PROGRAM Intfc_Upstream_ML
VAR
	Upstream_Upper_LaneA_Comm		: FB_ReadAdsSymByName;
	Upstream_Upper_LaneB_Comm		: FB_ReadAdsSymByName;
	Upstream_Upper_ExitLane_Comm	: FB_ReadAdsSymByName;
	Upstream_Lower_LaneA_Comm		: FB_ReadAdsSymByName;
	Upstream_Lower_LaneB_Comm		: FB_ReadAdsSymByName;
	Upstream_Lower_ExitLane_Comm	: FB_ReadAdsSymByName;
	UpdateRate						: TIME;
	UpdateTimer						: TON;
	UpdateCounter					: CTU;
END_VAR

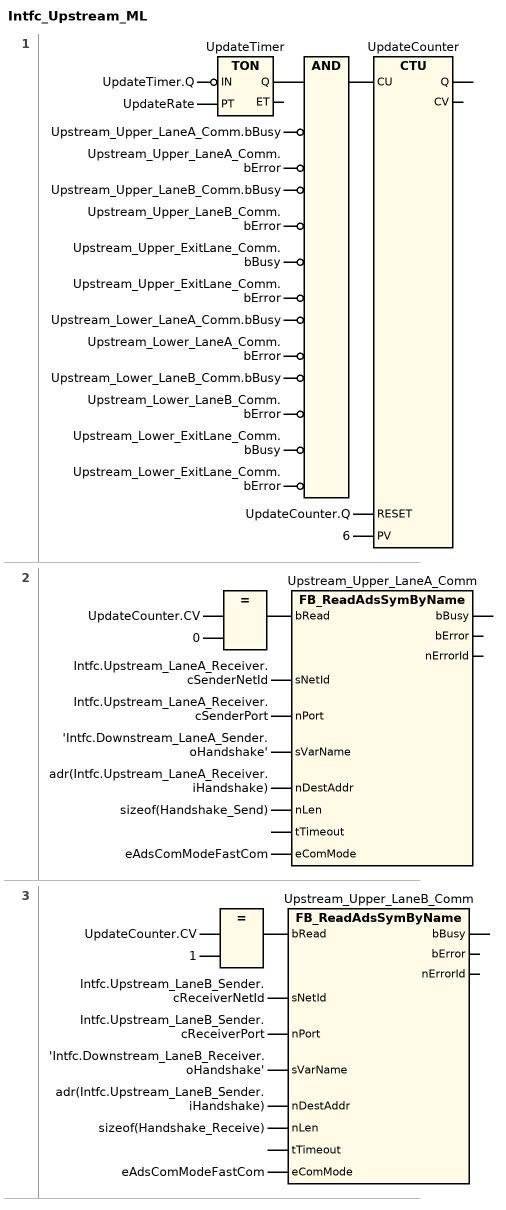
// NETWORK 1
UpdateTimer(IN := NOT UpdateTimer.Q, PT := UpdateRate); // TON
UpdateCounter(
    CU := UpdateTimer.Q AND NOT Upstream_Upper_LaneA_Comm.bBusy AND NOT Upstream_Upper_LaneA_Comm.bError AND NOT Upstream_Upper_LaneB_Comm.bBusy AND NOT Upstream_Upper_LaneB_Comm.bError AND NOT Upstream_Upper_ExitLane_Comm.bBusy AND NOT Upstream_Upper_ExitLane_Comm.bError AND NOT Upstream_Lower_LaneA_Comm.bBusy AND NOT Upstream_Lower_LaneA_Comm.bError AND NOT Upstream_Lower_LaneB_Comm.bBusy AND NOT Upstream_Lower_LaneB_Comm.bError AND NOT Upstream_Lower_ExitLane_Comm.bBusy AND NOT Upstream_Lower_ExitLane_Comm.bError,
    RESET := UpdateCounter.Q,
    PV := 6); // CTU

// NETWORK 2
Upstream_Upper_LaneA_Comm(
    bRead := UpdateCounter.CV = 0,
    sNetId := Intfc.Upstream_LaneA_Receiver.cSenderNetId,
    nPort := Intfc.Upstream_LaneA_Receiver.cSenderPort,
    sVarName := 'Intfc.Downstream_LaneA_Sender.oHandshake',
    nDestAddr := adr(Intfc.Upstream_LaneA_Receiver.iHandshake),
    nLen := sizeof(Handshake_Send),
    eComMode := eAdsComModeFastCom); // FB_ReadAdsSymByName

// NETWORK 3
Upstream_Upper_LaneB_Comm(
    bRead := UpdateCounter.CV = 1,
    sNetId := Intfc.Upstream_LaneB_Sender.cReceiverNetId,
    nPort := Intfc.Upstream_LaneB_Sender.cReceiverPort,
    sVarName := 'Intfc.Downstream_LaneB_Receiver.oHandshake',
    nDestAddr := adr(Intfc.Upstream_LaneB_Sender.iHandshake),
    nLen := sizeof(Handshake_Receive),
    eComMode := eAdsComModeFastCom); // FB_ReadAdsSymByName

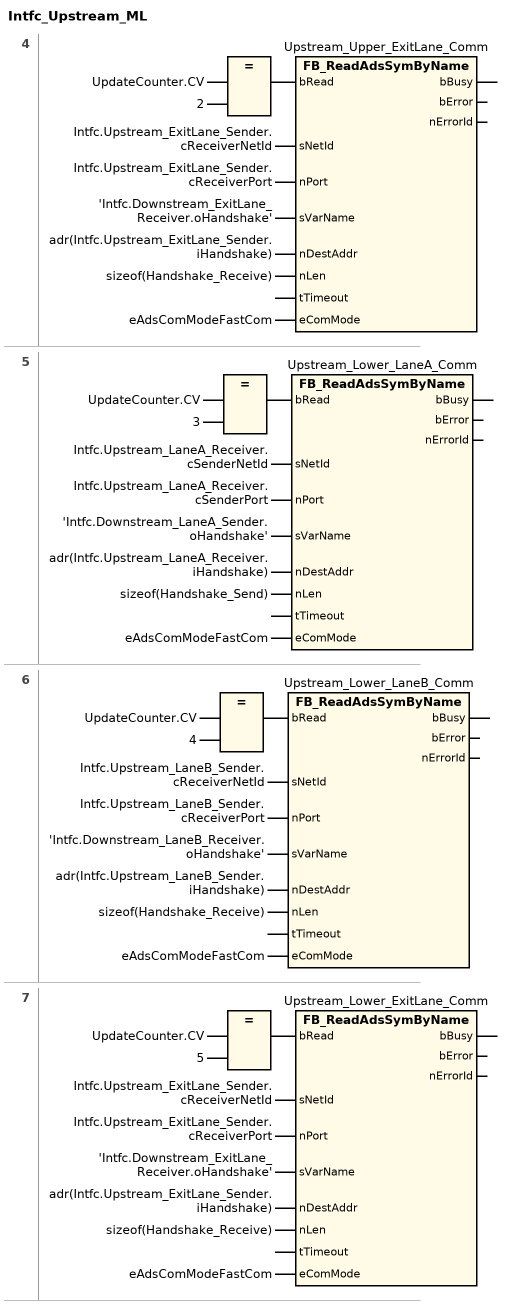
// NETWORK 4
Upstream_Upper_ExitLane_Comm(
    bRead := UpdateCounter.CV = 2,
    sNetId := Intfc.Upstream_ExitLane_Sender.cReceiverNetId,
    nPort := Intfc.Upstream_ExitLane_Sender.cReceiverPort,
    sVarName := 'Intfc.Downstream_ExitLane_Receiver.oHandshake',
    nDestAddr := adr(Intfc.Upstream_ExitLane_Sender.iHandshake),
    nLen := sizeof(Handshake_Receive),
    eComMode := eAdsComModeFastCom); // FB_ReadAdsSymByName

// NETWORK 5
Upstream_Lower_LaneA_Comm(
    bRead := UpdateCounter.CV = 3,
    sNetId := Intfc.Upstream_LaneA_Receiver.cSenderNetId,
    nPort := Intfc.Upstream_LaneA_Receiver.cSenderPort,
    sVarName := 'Intfc.Downstream_LaneA_Sender.oHandshake',
    nDestAddr := adr(Intfc.Upstream_LaneA_Receiver.iHandshake),
    nLen := sizeof(Handshake_Send),
    eComMode := eAdsComModeFastCom); // FB_ReadAdsSymByName

// NETWORK 6
Upstream_Lower_LaneB_Comm(
    bRead := UpdateCounter.CV = 4,
    sNetId := Intfc.Upstream_LaneB_Sender.cReceiverNetId,
    nPort := Intfc.Upstream_LaneB_Sender.cReceiverPort,
    sVarName := 'Intfc.Downstream_LaneB_Receiver.oHandshake',
    nDestAddr := adr(Intfc.Upstream_LaneB_Sender.iHandshake),
    nLen := sizeof(Handshake_Receive),
    eComMode := eAdsComModeFastCom); // FB_ReadAdsSymByName

// NETWORK 7
Upstream_Lower_ExitLane_Comm(
    bRead := UpdateCounter.CV = 5,
    sNetId := Intfc.Upstream_ExitLane_Sender.cReceiverNetId,
    nPort := Intfc.Upstream_ExitLane_Sender.cReceiverPort,
    sVarName := 'Intfc.Downstream_ExitLane_Receiver.oHandshake',
    nDestAddr := adr(Intfc.Upstream_ExitLane_Sender.iHandshake),
    nLen := sizeof(Handshake_Receive),
    eComMode := eAdsComModeFastCom); // FB_ReadAdsSymByName

END_PROGRAM

(* stored: Version 1.1.0.1, ProductVersion 3.1.4022.11
   POU Intfc_Upstream_ML: Id {7d1cbfeb-5ff5-4a3e-b870-a211d24d39db}, SpecialFunc None *)
